PROGRAM BeamEnChain
VAR
	BeamEn	AT %Q*:BOOL;
END_VAR

BeamEn := TRUE;

END_PROGRAM

(* stored: Version 1.1.0.1, ProductVersion 3.1.4022.10
   POU BeamEnChain: Id {51346549-1d7f-4261-9944-e59c41e34fe8}, SpecialFunc None *)
